// TIA Portal V20 export
DATA_BLOCK "ReelCutToStack40"   // DB223
// stored: InstanceOfName typeReelCutToStack, InstanceOfType UDT
"typeReelCutToStack"
   // VAR
   //    Load_Enable : Bool;
   //    Load_Complete_Comfirm : Bool;
   //    Cell_Data_Report : Bool;
   //    signal3 : Bool;
   //    signal4 : Bool;
   //    signal5 : Bool;
   //    signal6 : Bool;
   //    signal7 : Bool;
   //    signal8 : Bool;
   //    signal9 : Bool;
   //    signal10 : Bool;
   //    signal11 : Bool;
   //    signal12 : Bool;
   //    signal13 : Bool;
   //    signal14 : Bool;
   //    HeartBeat : Bool;
   //    signal16 : Bool;
   //    signal17 : Bool;
   //    signal18 : Bool;
   //    signal19 : Bool;
   //    signal20 : Bool;
   //    signal21 : Bool;
   //    signal22 : Bool;
   //    signal23 : Bool;
   //    signal24 : Bool;
   //    signal25 : Bool;
   //    signal26 : Bool;
   //    signal27 : Bool;
   //    signal28 : Bool;
   //    signal29 : Bool;
   //    signal30 : Bool;
   //    signal31 : Bool;
   //    signal32 : Bool;
   //    signal33 : Bool;
   //    signal34 : Bool;
   //    signal35 : Bool;
   //    signal36 : Bool;
   //    signal37 : Bool;
   //    signal38 : Bool;
   //    signal39 : Bool;
   //    signal40 : Bool;
   //    signal41 : Bool;
   //    signal42 : Bool;
   //    signal43 : Bool;
   //    signal44 : Bool;
   //    signal45 : Bool;
   //    signal46 : Bool;
   //    signal47 : Bool;
   //    signal48 : Bool;
   //    signal49 : Bool;
   //    signal50 : Bool;
   //    signal51 : Bool;
   //    signal52 : Bool;
   //    signal53 : Bool;
   //    signal54 : Bool;
   //    signal55 : Bool;
   //    signal56 : Bool;
   //    signal57 : Bool;
   //    signal58 : Bool;
   //    signal59 : Bool;
   //    signal60 : Bool;
   //    signal61 : Bool;
   //    signal62 : Bool;
   //    signal63 : Bool;
   //    signal64 : Bool;
   //    signal65 : Bool;
   //    signal66 : Bool;
   //    signal67 : Bool;
   //    signal68 : Bool;
   //    signal69 : Bool;
   //    signal70 : Bool;
   //    signal71 : Bool;
   //    signal72 : Bool;
   //    signal73 : Bool;
   //    signal74 : Bool;
   //    signal75 : Bool;
   //    signal76 : Bool;
   //    signal77 : Bool;
   //    signal78 : Bool;
   //    signal79 : Bool;
   //    signal80 : Bool;
   //    signal81 : Bool;
   //    signal82 : Bool;
   //    signal83 : Bool;
   //    signal84 : Bool;
   //    signal85 : Bool;
   //    signal86 : Bool;
   //    signal87 : Bool;
   //    signal88 : Bool;
   //    signal89 : Bool;
   //    signal90 : Bool;
   //    signal91 : Bool;
   //    signal92 : Bool;
   //    signal93 : Bool;
   //    signal94 : Bool;
   //    signal95 : Bool;
   // END_VAR
BEGIN
END_DATA_BLOCK
